# EPICS autosave request: iocBoot/iocTune/auto_settings_tune.req
file "tune_settings.req",                P=$(P),  R=$(R)
